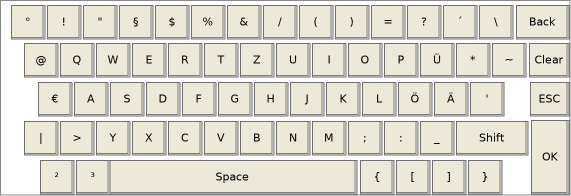
VISUALIZATION KeypadLayout  // 571x196
VAR_IN_OUT
	stVariableValue : STRING;
	bInit : BOOL;
	bShift : BOOL;
	stOutputValue : STRING;
	iCaretPosition	: INT;
	iSelectionStart	: INT;
	iSelectionEnd	: INT;
	flags: DWORD;
END_VAR
    Button (531,120 38x74), "OK"
        OnMouseDown: CloseDialog Dialog=Keypad, Result=OK, NumpadKeypad=True, NumpadKeypadSet=True
    Button (530,82 39x34), "ESC"
        OnMouseDown: CloseDialog Dialog=Keypad, Result=Cancel, NumpadKeypad=True, NumpadKeypadSet=True
    Button (529,43 40x34), "Clear"
        OnMouseDown: execute {
            stVariableValue := '';
            stOutputValue := '';
            iCaretPosition	:= 1;
            iSelectionStart	:= 1;
            iSelectionEnd := 1;
        }
    Button (516,5 53x34), "Back"
        OnMouseDown: execute { VisuDlg_ProcessBack(stOutputValue, stVariableValue, iCaretPosition, iSelectionStart, iSelectionEnd, bInit); }
    Button (456,121 72x34), "Shift"
        OnMouseDown: toggle bShift
    Button (108,160 249x34), "Space"
        OnMouseDown: execute { VisuDlg_ProcessChar(stOutputValue, stVariableValue, iCaretPosition, iSelectionStart, iSelectionEnd, (flags AND VisuElems.Visu_InputFlags.Password) = 1, ' '); }
    Button (40,160 34x34), "²"
        OnMouseDown: execute { VisuDlg_ProcessChar(stOutputValue, stVariableValue, iCaretPosition, iSelectionStart, iSelectionEnd, (flags AND VisuElems.Visu_InputFlags.Password) = 1, '²'); }
    Button (76,160 34x34), "³"
        OnMouseDown: execute { VisuDlg_ProcessChar(stOutputValue, stVariableValue, iCaretPosition, iSelectionStart, iSelectionEnd, (flags AND VisuElems.Visu_InputFlags.Password) = 1, '³'); }
    Button (360,160 34x34), "{"
        OnMouseDown: execute { VisuDlg_ProcessChar(stOutputValue, stVariableValue, iCaretPosition, iSelectionStart, iSelectionEnd, (flags AND VisuElems.Visu_InputFlags.Password) = 1, '{'); }
    Button (396,160 34x34), "["
        OnMouseDown: execute { VisuDlg_ProcessChar(stOutputValue, stVariableValue, iCaretPosition, iSelectionStart, iSelectionEnd, (flags AND VisuElems.Visu_InputFlags.Password) = 1, '['); }
    Button (432,160 34x34), "]"
        OnMouseDown: execute { VisuDlg_ProcessChar(stOutputValue, stVariableValue, iCaretPosition, iSelectionStart, iSelectionEnd, (flags AND VisuElems.Visu_InputFlags.Password) = 1, ']'); }
    Button (468,160 34x34), "}"
        OnMouseDown: execute { VisuDlg_ProcessChar(stOutputValue, stVariableValue, iCaretPosition, iSelectionStart, iSelectionEnd, (flags AND VisuElems.Visu_InputFlags.Password) = 1, '}'); }
    Button (24,121 34x34), "|"
        OnMouseDown: execute { VisuDlg_ProcessChar(stOutputValue, stVariableValue, iCaretPosition, iSelectionStart, iSelectionEnd, (flags AND VisuElems.Visu_InputFlags.Password) = 1, '|'); }
    Button (60,121 34x34), "<", invisible if: NOT bShift
        OnMouseDown: execute { VisuDlg_ProcessChar(stOutputValue, stVariableValue, iCaretPosition, iSelectionStart, iSelectionEnd, (flags AND VisuElems.Visu_InputFlags.Password) = 1, '<'); }
    Button (60,121 34x34), ">", invisible if: bShift
        OnMouseDown: execute { VisuDlg_ProcessChar(stOutputValue, stVariableValue, iCaretPosition, iSelectionStart, iSelectionEnd, (flags AND VisuElems.Visu_InputFlags.Password) = 1, '>'); }
    Button (96,121 34x34), "y", invisible if: NOT bShift
        OnMouseDown: execute { VisuDlg_ProcessChar(stOutputValue, stVariableValue, iCaretPosition, iSelectionStart, iSelectionEnd, (flags AND VisuElems.Visu_InputFlags.Password) = 1, 'y'); }
    Button (96,121 34x34), "Y", invisible if: bShift
        OnMouseDown: execute { VisuDlg_ProcessChar(stOutputValue, stVariableValue, iCaretPosition, iSelectionStart, iSelectionEnd, (flags AND VisuElems.Visu_InputFlags.Password) = 1, 'Y'); }
    Button (132,121 34x34), "x", invisible if: NOT bShift
        OnMouseDown: execute { VisuDlg_ProcessChar(stOutputValue, stVariableValue, iCaretPosition, iSelectionStart, iSelectionEnd, (flags AND VisuElems.Visu_InputFlags.Password) = 1, 'x'); }
    Button (132,121 34x34), "X", invisible if: bShift
        OnMouseDown: execute { VisuDlg_ProcessChar(stOutputValue, stVariableValue, iCaretPosition, iSelectionStart, iSelectionEnd, (flags AND VisuElems.Visu_InputFlags.Password) = 1, 'X'); }
    Button (168,121 34x34), "c", invisible if: NOT bShift
        OnMouseDown: execute { VisuDlg_ProcessChar(stOutputValue, stVariableValue, iCaretPosition, iSelectionStart, iSelectionEnd, (flags AND VisuElems.Visu_InputFlags.Password) = 1, 'c'); }
    Button (168,121 34x34), "C", invisible if: bShift
        OnMouseDown: execute { VisuDlg_ProcessChar(stOutputValue, stVariableValue, iCaretPosition, iSelectionStart, iSelectionEnd, (flags AND VisuElems.Visu_InputFlags.Password) = 1, 'C'); }
    Button (204,121 34x34), "v", invisible if: NOT bShift
        OnMouseDown: execute { VisuDlg_ProcessChar(stOutputValue, stVariableValue, iCaretPosition, iSelectionStart, iSelectionEnd, (flags AND VisuElems.Visu_InputFlags.Password) = 1, 'v'); }
    Button (204,121 34x34), "V", invisible if: bShift
        OnMouseDown: execute { VisuDlg_ProcessChar(stOutputValue, stVariableValue, iCaretPosition, iSelectionStart, iSelectionEnd, (flags AND VisuElems.Visu_InputFlags.Password) = 1, 'V'); }
    Button (240,121 34x34), "b", invisible if: NOT bShift
        OnMouseDown: execute { VisuDlg_ProcessChar(stOutputValue, stVariableValue, iCaretPosition, iSelectionStart, iSelectionEnd, (flags AND VisuElems.Visu_InputFlags.Password) = 1, 'b'); }
    Button (240,121 34x34), "B", invisible if: bShift
        OnMouseDown: execute { VisuDlg_ProcessChar(stOutputValue, stVariableValue, iCaretPosition, iSelectionStart, iSelectionEnd, (flags AND VisuElems.Visu_InputFlags.Password) = 1, 'B'); }
    Button (276,121 34x34), "n", invisible if: NOT bShift
        OnMouseDown: execute { VisuDlg_ProcessChar(stOutputValue, stVariableValue, iCaretPosition, iSelectionStart, iSelectionEnd, (flags AND VisuElems.Visu_InputFlags.Password) = 1, 'n'); }
    Button (276,121 34x34), "N", invisible if: bShift
        OnMouseDown: execute { VisuDlg_ProcessChar(stOutputValue, stVariableValue, iCaretPosition, iSelectionStart, iSelectionEnd, (flags AND VisuElems.Visu_InputFlags.Password) = 1, 'N'); }
    Button (312,121 34x34), "m", invisible if: NOT bShift
        OnMouseDown: execute { VisuDlg_ProcessChar(stOutputValue, stVariableValue, iCaretPosition, iSelectionStart, iSelectionEnd, (flags AND VisuElems.Visu_InputFlags.Password) = 1, 'm'); }
    Button (312,121 34x34), "M", invisible if: bShift
        OnMouseDown: execute { VisuDlg_ProcessChar(stOutputValue, stVariableValue, iCaretPosition, iSelectionStart, iSelectionEnd, (flags AND VisuElems.Visu_InputFlags.Password) = 1, 'M'); }
    Button (348,121 34x34), ",", invisible if: NOT bShift
        OnMouseDown: execute { VisuDlg_ProcessChar(stOutputValue, stVariableValue, iCaretPosition, iSelectionStart, iSelectionEnd, (flags AND VisuElems.Visu_InputFlags.Password) = 1, ','); }
    Button (348,121 34x34), ";", invisible if: bShift
        OnMouseDown: execute { VisuDlg_ProcessChar(stOutputValue, stVariableValue, iCaretPosition, iSelectionStart, iSelectionEnd, (flags AND VisuElems.Visu_InputFlags.Password) = 1, ';'); }
    Button (384,121 34x34), ".", invisible if: NOT bShift
        OnMouseDown: execute { VisuDlg_ProcessChar(stOutputValue, stVariableValue, iCaretPosition, iSelectionStart, iSelectionEnd, (flags AND VisuElems.Visu_InputFlags.Password) = 1, '.'); }
    Button (384,121 34x34), ":", invisible if: bShift
        OnMouseDown: execute { VisuDlg_ProcessChar(stOutputValue, stVariableValue, iCaretPosition, iSelectionStart, iSelectionEnd, (flags AND VisuElems.Visu_InputFlags.Password) = 1, ':'); }
    Button (420,121 34x34), "-", invisible if: NOT bShift
        OnMouseDown: execute { VisuDlg_ProcessChar(stOutputValue, stVariableValue, iCaretPosition, iSelectionStart, iSelectionEnd, (flags AND VisuElems.Visu_InputFlags.Password) = 1, '-'); }
    Button (420,121 34x34), "_", invisible if: bShift
        OnMouseDown: execute { VisuDlg_ProcessChar(stOutputValue, stVariableValue, iCaretPosition, iSelectionStart, iSelectionEnd, (flags AND VisuElems.Visu_InputFlags.Password) = 1, '_'); }
    Button (38,82 34x34), "€"
        OnMouseDown: execute { VisuDlg_ProcessChar(stOutputValue, stVariableValue, iCaretPosition, iSelectionStart, iSelectionEnd, (flags AND VisuElems.Visu_InputFlags.Password) = 1, '€'); }
    Button (74,82 34x34), "a", invisible if: NOT bShift
        OnMouseDown: execute { VisuDlg_ProcessChar(stOutputValue, stVariableValue, iCaretPosition, iSelectionStart, iSelectionEnd, (flags AND VisuElems.Visu_InputFlags.Password) = 1, 'a'); }
    Button (74,82 34x34), "A", invisible if: bShift
        OnMouseDown: execute { VisuDlg_ProcessChar(stOutputValue, stVariableValue, iCaretPosition, iSelectionStart, iSelectionEnd, (flags AND VisuElems.Visu_InputFlags.Password) = 1, 'A'); }
    Button (110,82 34x34), "s", invisible if: NOT bShift
        OnMouseDown: execute { VisuDlg_ProcessChar(stOutputValue, stVariableValue, iCaretPosition, iSelectionStart, iSelectionEnd, (flags AND VisuElems.Visu_InputFlags.Password) = 1, 's'); }
    Button (110,82 34x34), "S", invisible if: bShift
        OnMouseDown: execute { VisuDlg_ProcessChar(stOutputValue, stVariableValue, iCaretPosition, iSelectionStart, iSelectionEnd, (flags AND VisuElems.Visu_InputFlags.Password) = 1, 'S'); }
    Button (146,82 34x34), "d", invisible if: NOT bShift
        OnMouseDown: execute { VisuDlg_ProcessChar(stOutputValue, stVariableValue, iCaretPosition, iSelectionStart, iSelectionEnd, (flags AND VisuElems.Visu_InputFlags.Password) = 1, 'd'); }
    Button (146,82 34x34), "D", invisible if: bShift
        OnMouseDown: execute { VisuDlg_ProcessChar(stOutputValue, stVariableValue, iCaretPosition, iSelectionStart, iSelectionEnd, (flags AND VisuElems.Visu_InputFlags.Password) = 1, 'D'); }
    Button (182,82 34x34), "f", invisible if: NOT bShift
        OnMouseDown: execute { VisuDlg_ProcessChar(stOutputValue, stVariableValue, iCaretPosition, iSelectionStart, iSelectionEnd, (flags AND VisuElems.Visu_InputFlags.Password) = 1, 'f'); }
    Button (182,82 34x34), "F", invisible if: bShift
        OnMouseDown: execute { VisuDlg_ProcessChar(stOutputValue, stVariableValue, iCaretPosition, iSelectionStart, iSelectionEnd, (flags AND VisuElems.Visu_InputFlags.Password) = 1, 'F'); }
    Button (218,82 34x34), "g", invisible if: NOT bShift
        OnMouseDown: execute { VisuDlg_ProcessChar(stOutputValue, stVariableValue, iCaretPosition, iSelectionStart, iSelectionEnd, (flags AND VisuElems.Visu_InputFlags.Password) = 1, 'g'); }
    Button (218,82 34x34), "G", invisible if: bShift
        OnMouseDown: execute { VisuDlg_ProcessChar(stOutputValue, stVariableValue, iCaretPosition, iSelectionStart, iSelectionEnd, (flags AND VisuElems.Visu_InputFlags.Password) = 1, 'G'); }
    Button (254,82 34x34), "h", invisible if: NOT bShift
        OnMouseDown: execute { VisuDlg_ProcessChar(stOutputValue, stVariableValue, iCaretPosition, iSelectionStart, iSelectionEnd, (flags AND VisuElems.Visu_InputFlags.Password) = 1, 'h'); }
    Button (254,82 34x34), "H", invisible if: bShift
        OnMouseDown: execute { VisuDlg_ProcessChar(stOutputValue, stVariableValue, iCaretPosition, iSelectionStart, iSelectionEnd, (flags AND VisuElems.Visu_InputFlags.Password) = 1, 'H'); }
    Button (290,82 34x34), "j", invisible if: NOT bShift
        OnMouseDown: execute { VisuDlg_ProcessChar(stOutputValue, stVariableValue, iCaretPosition, iSelectionStart, iSelectionEnd, (flags AND VisuElems.Visu_InputFlags.Password) = 1, 'j'); }
    Button (290,82 34x34), "J", invisible if: bShift
        OnMouseDown: execute { VisuDlg_ProcessChar(stOutputValue, stVariableValue, iCaretPosition, iSelectionStart, iSelectionEnd, (flags AND VisuElems.Visu_InputFlags.Password) = 1, 'J'); }
    Button (326,82 34x34), "k", invisible if: NOT bShift
        OnMouseDown: execute { VisuDlg_ProcessChar(stOutputValue, stVariableValue, iCaretPosition, iSelectionStart, iSelectionEnd, (flags AND VisuElems.Visu_InputFlags.Password) = 1, 'k'); }
    Button (326,82 34x34), "K", invisible if: bShift
        OnMouseDown: execute { VisuDlg_ProcessChar(stOutputValue, stVariableValue, iCaretPosition, iSelectionStart, iSelectionEnd, (flags AND VisuElems.Visu_InputFlags.Password) = 1, 'K'); }
    Button (362,82 34x34), "l", invisible if: NOT bShift
        OnMouseDown: execute { VisuDlg_ProcessChar(stOutputValue, stVariableValue, iCaretPosition, iSelectionStart, iSelectionEnd, (flags AND VisuElems.Visu_InputFlags.Password) = 1, 'l'); }
    Button (362,82 34x34), "L", invisible if: bShift
        OnMouseDown: execute { VisuDlg_ProcessChar(stOutputValue, stVariableValue, iCaretPosition, iSelectionStart, iSelectionEnd, (flags AND VisuElems.Visu_InputFlags.Password) = 1, 'L'); }
    Button (398,82 34x34), "ö", invisible if: NOT bShift
        OnMouseDown: execute { VisuDlg_ProcessChar(stOutputValue, stVariableValue, iCaretPosition, iSelectionStart, iSelectionEnd, (flags AND VisuElems.Visu_InputFlags.Password) = 1, 'ö'); }
    Button (398,82 34x34), "Ö", invisible if: bShift
        OnMouseDown: execute { VisuDlg_ProcessChar(stOutputValue, stVariableValue, iCaretPosition, iSelectionStart, iSelectionEnd, (flags AND VisuElems.Visu_InputFlags.Password) = 1, 'Ö'); }
    Button (434,82 34x34), "ä", invisible if: NOT bShift
        OnMouseDown: execute { VisuDlg_ProcessChar(stOutputValue, stVariableValue, iCaretPosition, iSelectionStart, iSelectionEnd, (flags AND VisuElems.Visu_InputFlags.Password) = 1, 'ä'); }
    Button (434,82 34x34), "Ä", invisible if: bShift
        OnMouseDown: execute { VisuDlg_ProcessChar(stOutputValue, stVariableValue, iCaretPosition, iSelectionStart, iSelectionEnd, (flags AND VisuElems.Visu_InputFlags.Password) = 1, 'Ä'); }
    Button (470,82 34x34), "#", invisible if: NOT bShift
        OnMouseDown: execute { VisuDlg_ProcessChar(stOutputValue, stVariableValue, iCaretPosition, iSelectionStart, iSelectionEnd, (flags AND VisuElems.Visu_InputFlags.Password) = 1, '#'); }
    Button (470,82 34x34), "'", invisible if: bShift
        OnMouseDown: execute { VisuDlg_ProcessChar(stOutputValue, stVariableValue, iCaretPosition, iSelectionStart, iSelectionEnd, (flags AND VisuElems.Visu_InputFlags.Password) = 1, '$''); }
    Button (24,43 34x34), "@"
        OnMouseDown: execute { VisuDlg_ProcessChar(stOutputValue, stVariableValue, iCaretPosition, iSelectionStart, iSelectionEnd, (flags AND VisuElems.Visu_InputFlags.Password) = 1, '@'); }
    Button (60,43 34x34), "q", invisible if: NOT bShift
        OnMouseDown: execute { VisuDlg_ProcessChar(stOutputValue, stVariableValue, iCaretPosition, iSelectionStart, iSelectionEnd, (flags AND VisuElems.Visu_InputFlags.Password) = 1, 'q'); }
    Button (60,43 34x34), "Q", invisible if: bShift
        OnMouseDown: execute { VisuDlg_ProcessChar(stOutputValue, stVariableValue, iCaretPosition, iSelectionStart, iSelectionEnd, (flags AND VisuElems.Visu_InputFlags.Password) = 1, 'Q'); }
    Button (96,43 34x34), "w", invisible if: NOT bShift
        OnMouseDown: execute { VisuDlg_ProcessChar(stOutputValue, stVariableValue, iCaretPosition, iSelectionStart, iSelectionEnd, (flags AND VisuElems.Visu_InputFlags.Password) = 1, 'w'); }
    Button (96,43 34x34), "W", invisible if: bShift
        OnMouseDown: execute { VisuDlg_ProcessChar(stOutputValue, stVariableValue, iCaretPosition, iSelectionStart, iSelectionEnd, (flags AND VisuElems.Visu_InputFlags.Password) = 1, 'W'); }
    Button (132,43 34x34), "e", invisible if: NOT bShift
        OnMouseDown: execute { VisuDlg_ProcessChar(stOutputValue, stVariableValue, iCaretPosition, iSelectionStart, iSelectionEnd, (flags AND VisuElems.Visu_InputFlags.Password) = 1, 'e'); }
    Button (132,43 34x34), "E", invisible if: bShift
        OnMouseDown: execute { VisuDlg_ProcessChar(stOutputValue, stVariableValue, iCaretPosition, iSelectionStart, iSelectionEnd, (flags AND VisuElems.Visu_InputFlags.Password) = 1, 'E'); }
    Button (168,43 34x34), "r", invisible if: NOT bShift
        OnMouseDown: execute { VisuDlg_ProcessChar(stOutputValue, stVariableValue, iCaretPosition, iSelectionStart, iSelectionEnd, (flags AND VisuElems.Visu_InputFlags.Password) = 1, 'r'); }
    Button (168,43 34x34), "R", invisible if: bShift
        OnMouseDown: execute { VisuDlg_ProcessChar(stOutputValue, stVariableValue, iCaretPosition, iSelectionStart, iSelectionEnd, (flags AND VisuElems.Visu_InputFlags.Password) = 1, 'R'); }
    Button (204,43 34x34), "t", invisible if: NOT bShift
        OnMouseDown: execute { VisuDlg_ProcessChar(stOutputValue, stVariableValue, iCaretPosition, iSelectionStart, iSelectionEnd, (flags AND VisuElems.Visu_InputFlags.Password) = 1, 't'); }
    Button (204,43 34x34), "T", invisible if: bShift
        OnMouseDown: execute { VisuDlg_ProcessChar(stOutputValue, stVariableValue, iCaretPosition, iSelectionStart, iSelectionEnd, (flags AND VisuElems.Visu_InputFlags.Password) = 1, 'T'); }
    Button (240,43 34x34), "z", invisible if: NOT bShift
        OnMouseDown: execute { VisuDlg_ProcessChar(stOutputValue, stVariableValue, iCaretPosition, iSelectionStart, iSelectionEnd, (flags AND VisuElems.Visu_InputFlags.Password) = 1, 'z'); }
    Button (240,43 34x34), "Z", invisible if: bShift
        OnMouseDown: execute { VisuDlg_ProcessChar(stOutputValue, stVariableValue, iCaretPosition, iSelectionStart, iSelectionEnd, (flags AND VisuElems.Visu_InputFlags.Password) = 1, 'Z'); }
    Button (276,43 34x34), "u", invisible if: NOT bShift
        OnMouseDown: execute { VisuDlg_ProcessChar(stOutputValue, stVariableValue, iCaretPosition, iSelectionStart, iSelectionEnd, (flags AND VisuElems.Visu_InputFlags.Password) = 1, 'u'); }
    Button (276,43 34x34), "U", invisible if: bShift
        OnMouseDown: execute { VisuDlg_ProcessChar(stOutputValue, stVariableValue, iCaretPosition, iSelectionStart, iSelectionEnd, (flags AND VisuElems.Visu_InputFlags.Password) = 1, 'U'); }
    Button (312,43 34x34), "i", invisible if: NOT bShift
        OnMouseDown: execute { VisuDlg_ProcessChar(stOutputValue, stVariableValue, iCaretPosition, iSelectionStart, iSelectionEnd, (flags AND VisuElems.Visu_InputFlags.Password) = 1, 'i'); }
    Button (312,43 34x34), "I", invisible if: bShift
        OnMouseDown: execute { VisuDlg_ProcessChar(stOutputValue, stVariableValue, iCaretPosition, iSelectionStart, iSelectionEnd, (flags AND VisuElems.Visu_InputFlags.Password) = 1, 'I'); }
    Button (348,43 34x34), "o", invisible if: NOT bShift
        OnMouseDown: execute { VisuDlg_ProcessChar(stOutputValue, stVariableValue, iCaretPosition, iSelectionStart, iSelectionEnd, (flags AND VisuElems.Visu_InputFlags.Password) = 1, 'o'); }
    Button (348,43 34x34), "O", invisible if: bShift
        OnMouseDown: execute { VisuDlg_ProcessChar(stOutputValue, stVariableValue, iCaretPosition, iSelectionStart, iSelectionEnd, (flags AND VisuElems.Visu_InputFlags.Password) = 1, 'O'); }
    Button (384,43 34x34), "p", invisible if: NOT bShift
        OnMouseDown: execute { VisuDlg_ProcessChar(stOutputValue, stVariableValue, iCaretPosition, iSelectionStart, iSelectionEnd, (flags AND VisuElems.Visu_InputFlags.Password) = 1, 'p'); }
    Button (384,43 34x34), "P", invisible if: bShift
        OnMouseDown: execute { VisuDlg_ProcessChar(stOutputValue, stVariableValue, iCaretPosition, iSelectionStart, iSelectionEnd, (flags AND VisuElems.Visu_InputFlags.Password) = 1, 'P'); }
    Button (420,43 34x34), "ü", invisible if: NOT bShift
        OnMouseDown: execute { VisuDlg_ProcessChar(stOutputValue, stVariableValue, iCaretPosition, iSelectionStart, iSelectionEnd, (flags AND VisuElems.Visu_InputFlags.Password) = 1, 'ü'); }
    Button (420,43 34x34), "Ü", invisible if: bShift
        OnMouseDown: execute { VisuDlg_ProcessChar(stOutputValue, stVariableValue, iCaretPosition, iSelectionStart, iSelectionEnd, (flags AND VisuElems.Visu_InputFlags.Password) = 1, 'Ü'); }
    Button (456,43 34x34), "+", invisible if: NOT bShift
        OnMouseDown: execute { VisuDlg_ProcessChar(stOutputValue, stVariableValue, iCaretPosition, iSelectionStart, iSelectionEnd, (flags AND VisuElems.Visu_InputFlags.Password) = 1, '+'); }
    Button (456,43 34x34), "*", invisible if: bShift
        OnMouseDown: execute { VisuDlg_ProcessChar(stOutputValue, stVariableValue, iCaretPosition, iSelectionStart, iSelectionEnd, (flags AND VisuElems.Visu_InputFlags.Password) = 1, '*'); }
    Button (492,43 34x34), "~"
        OnMouseDown: execute { VisuDlg_ProcessChar(stOutputValue, stVariableValue, iCaretPosition, iSelectionStart, iSelectionEnd, (flags AND VisuElems.Visu_InputFlags.Password) = 1, '~'); }
    Button (11,5 34x34), "^", invisible if: NOT bShift
        OnMouseDown: execute { VisuDlg_ProcessChar(stOutputValue, stVariableValue, iCaretPosition, iSelectionStart, iSelectionEnd, (flags AND VisuElems.Visu_InputFlags.Password) = 1, '^'); }
    Button (11,5 34x34), "°", invisible if: bShift
        OnMouseDown: execute { VisuDlg_ProcessChar(stOutputValue, stVariableValue, iCaretPosition, iSelectionStart, iSelectionEnd, (flags AND VisuElems.Visu_InputFlags.Password) = 1, '°'); }
    Button (47,5 34x34), "1", invisible if: NOT bShift
        OnMouseDown: execute { VisuDlg_ProcessChar(stOutputValue, stVariableValue, iCaretPosition, iSelectionStart, iSelectionEnd, (flags AND VisuElems.Visu_InputFlags.Password) = 1, '1'); }
    Button (47,5 34x34), "!", invisible if: bShift
        OnMouseDown: execute { VisuDlg_ProcessChar(stOutputValue, stVariableValue, iCaretPosition, iSelectionStart, iSelectionEnd, (flags AND VisuElems.Visu_InputFlags.Password) = 1, '!'); }
    Button (83,5 34x34), "2", invisible if: NOT bShift
        OnMouseDown: execute { VisuDlg_ProcessChar(stOutputValue, stVariableValue, iCaretPosition, iSelectionStart, iSelectionEnd, (flags AND VisuElems.Visu_InputFlags.Password) = 1, '2'); }
    Button (83,5 34x34), """, invisible if: bShift
        OnMouseDown: execute { VisuDlg_ProcessChar(stOutputValue, stVariableValue, iCaretPosition, iSelectionStart, iSelectionEnd, (flags AND VisuElems.Visu_InputFlags.Password) = 1, '"'); }
    Button (119,5 34x34), "3", invisible if: NOT bShift
        OnMouseDown: execute { VisuDlg_ProcessChar(stOutputValue, stVariableValue, iCaretPosition, iSelectionStart, iSelectionEnd, (flags AND VisuElems.Visu_InputFlags.Password) = 1, '3'); }
    Button (119,5 34x34), "§", invisible if: bShift
        OnMouseDown: execute { VisuDlg_ProcessChar(stOutputValue, stVariableValue, iCaretPosition, iSelectionStart, iSelectionEnd, (flags AND VisuElems.Visu_InputFlags.Password) = 1, '§'); }
    Button (155,5 34x34), "4", invisible if: NOT bShift
        OnMouseDown: execute { VisuDlg_ProcessChar(stOutputValue, stVariableValue, iCaretPosition, iSelectionStart, iSelectionEnd, (flags AND VisuElems.Visu_InputFlags.Password) = 1, '4'); }
    Button (155,5 34x34), "$", invisible if: bShift
        OnMouseDown: execute { VisuDlg_ProcessChar(stOutputValue, stVariableValue, iCaretPosition, iSelectionStart, iSelectionEnd, (flags AND VisuElems.Visu_InputFlags.Password) = 1, '$$'); }
    Button (191,5 34x34), "5", invisible if: NOT bShift
        OnMouseDown: execute { VisuDlg_ProcessChar(stOutputValue, stVariableValue, iCaretPosition, iSelectionStart, iSelectionEnd, (flags AND VisuElems.Visu_InputFlags.Password) = 1, '5'); }
    Button (191,5 34x34), "%", invisible if: bShift
        OnMouseDown: execute { VisuDlg_ProcessChar(stOutputValue, stVariableValue, iCaretPosition, iSelectionStart, iSelectionEnd, (flags AND VisuElems.Visu_InputFlags.Password) = 1, '%'); }
    Button (227,5 34x34), "6", invisible if: NOT bShift
        OnMouseDown: execute { VisuDlg_ProcessChar(stOutputValue, stVariableValue, iCaretPosition, iSelectionStart, iSelectionEnd, (flags AND VisuElems.Visu_InputFlags.Password) = 1, '6'); }
    Button (227,5 34x34), "&", invisible if: bShift
        OnMouseDown: execute { VisuDlg_ProcessChar(stOutputValue, stVariableValue, iCaretPosition, iSelectionStart, iSelectionEnd, (flags AND VisuElems.Visu_InputFlags.Password) = 1, '&'); }
    Button (263,5 34x34), "7", invisible if: NOT bShift
        OnMouseDown: execute { VisuDlg_ProcessChar(stOutputValue, stVariableValue, iCaretPosition, iSelectionStart, iSelectionEnd, (flags AND VisuElems.Visu_InputFlags.Password) = 1, '7'); }
    Button (263,5 34x34), "/", invisible if: bShift
        OnMouseDown: execute { VisuDlg_ProcessChar(stOutputValue, stVariableValue, iCaretPosition, iSelectionStart, iSelectionEnd, (flags AND VisuElems.Visu_InputFlags.Password) = 1, '/'); }
    Button (299,5 34x34), "8", invisible if: NOT bShift
        OnMouseDown: execute { VisuDlg_ProcessChar(stOutputValue, stVariableValue, iCaretPosition, iSelectionStart, iSelectionEnd, (flags AND VisuElems.Visu_InputFlags.Password) = 1, '8'); }
    Button (299,5 34x34), "(", invisible if: bShift
        OnMouseDown: execute { VisuDlg_ProcessChar(stOutputValue, stVariableValue, iCaretPosition, iSelectionStart, iSelectionEnd, (flags AND VisuElems.Visu_InputFlags.Password) = 1, '('); }
    Button (335,5 34x34), "9", invisible if: NOT bShift
        OnMouseDown: execute { VisuDlg_ProcessChar(stOutputValue, stVariableValue, iCaretPosition, iSelectionStart, iSelectionEnd, (flags AND VisuElems.Visu_InputFlags.Password) = 1, '9'); }
    Button (335,5 34x34), ")", invisible if: bShift
        OnMouseDown: execute { VisuDlg_ProcessChar(stOutputValue, stVariableValue, iCaretPosition, iSelectionStart, iSelectionEnd, (flags AND VisuElems.Visu_InputFlags.Password) = 1, ')'); }
    Button (371,5 34x34), "0", invisible if: NOT bShift
        OnMouseDown: execute { VisuDlg_ProcessChar(stOutputValue, stVariableValue, iCaretPosition, iSelectionStart, iSelectionEnd, (flags AND VisuElems.Visu_InputFlags.Password) = 1, '0'); }
    Button (371,5 34x34), "=", invisible if: bShift
        OnMouseDown: execute { VisuDlg_ProcessChar(stOutputValue, stVariableValue, iCaretPosition, iSelectionStart, iSelectionEnd, (flags AND VisuElems.Visu_InputFlags.Password) = 1, '='); }
    Button (407,5 34x34), "ß", invisible if: NOT bShift
        OnMouseDown: execute { VisuDlg_ProcessChar(stOutputValue, stVariableValue, iCaretPosition, iSelectionStart, iSelectionEnd, (flags AND VisuElems.Visu_InputFlags.Password) = 1, 'ß'); }
    Button (407,5 34x34), "?", invisible if: bShift
        OnMouseDown: execute { VisuDlg_ProcessChar(stOutputValue, stVariableValue, iCaretPosition, iSelectionStart, iSelectionEnd, (flags AND VisuElems.Visu_InputFlags.Password) = 1, '?'); }
    Button (443,5 34x34), "´"
        OnMouseDown: execute { VisuDlg_ProcessChar(stOutputValue, stVariableValue, iCaretPosition, iSelectionStart, iSelectionEnd, (flags AND VisuElems.Visu_InputFlags.Password) = 1, '´'); }
    Button (479,5 34x34), "\"
        OnMouseDown: execute { VisuDlg_ProcessChar(stOutputValue, stVariableValue, iCaretPosition, iSelectionStart, iSelectionEnd, (flags AND VisuElems.Visu_InputFlags.Password) = 1, '\'); }
END_VISUALIZATION

(* stored: Version 1.1.0.1, ProductVersion 3.1.4024.2
   Visu KeypadLayout: Id {234eb5d8-67f3-42da-bfa3-98a813c2f2a7} *)
